{attribute 'qualified_only'}
{attribute 'strict'}
TYPE FileMemoryAction :
(
	UNLOCKED := 0,
  READ,
  WRITE
);
END_TYPE

(* stored: Version 1.1.0.1, ProductVersion 3.1.4022.12
   DUT FileMemoryAction: Id {caf165a9-cb64-467e-8b54-64c6e6d0da73} *)
